(* This function block is responsible for holding the internal state of the function block that
   has the different tests in it (i.e. test-FB). Every test-FB can have one or more tests, and
   each test can do one or more asserts.
*)
{attribute 'call_after_init'}
{attribute 'reflection'}
FUNCTION_BLOCK FB_TestFunctionBlock IMPLEMENTS I_TestFunctionBlock
VAR
    {attribute 'instance-path'}
    {attribute 'noinit'}
    InstancePath : Tc2_Utilities.T_MaxString;

    (* This is a interface-pointer to the child-object that inherits this object
       in order for us to have a reference to calling the actual execution of the
       tests *) 
    RunnableTest : I_RunnableTestFunctionBlock;

    NumberOfTests : UINT := 0;
    TestNames : ARRAY[1..100] OF Tc2_Utilities.T_MaxString;
    TestFailed : ARRAY[1..100] OF BOOL;
END_VAR

METHOD PUBLIC AddTest
VAR_INPUT
    TestName : T_MaxString;
END_VAR
VAR
    CounterTestName : UINT;
END_VAR
(* Check if the test name already exists *)
FOR CounterTestName := 1 TO NumberOfTests BY 1 DO
    IF TestNames[CounterTestName] = TestName THEN
        RETURN; // Found
    END_IF
END_FOR

(* Not found. Add it. *)
TestNames[CounterTestName] := TestName;
NumberOfTests := NumberOfTests + 1;
END_METHOD

METHOD PUBLIC GetAmountOfFailedTests : UINT
VAR
    Counter : UINT;
    FailedTestsCount : UINT;
END_VAR
IF NumberOfTests > 0 THEN
    FOR Counter := 1 TO GetAmountOfTests() BY 1 DO
        IF TestFailed[Counter] = TRUE THEN
            FailedTestsCount := FailedTestsCount + 1;
        END_IF
    END_FOR
END_IF

GetAmountOfFailedTests := FailedTestsCount;
END_METHOD

METHOD PUBLIC GetAmountOfSuccessfulTests : UINT
GetAmountOfSuccessfulTests := GetAmountOfTests() - GetAmountOfFailedTests();
END_METHOD

METHOD PUBLIC GetAmountOfTests : UINT
GetAmountOfTests := NumberOfTests;
END_METHOD

METHOD PUBLIC GetInstancePath : Tc2_Utilities.T_MaxString
GetInstancePath := InstancePath;
END_METHOD

METHOD GetRunnable : I_RunnableTestFunctionBlock
GetRunnable := RunnableTest;
END_METHOD

{attribute 'call_after_init'}
METHOD PRIVATE Initialize
IF GVL.TestFunctionBlockAssertRegistered THEN
    GVL.AmountOfInitializedTestFunctionBlocks := GVL.AmountOfInitializedTestFunctionBlocks + 1;	
    GVL.TestFunctionBlockAddressess[GVL.AmountOfInitializedTestFunctionBlocks] := THIS^;
    GVL.TestFunctionBlockAssertRegistered := FALSE;
END_IF
END_METHOD

METHOD PUBLIC RegisterTestFunctionBlock
VAR_INPUT
	RunnableTestFunctionBlock : I_RunnableTestFunctionBlock;
END_VAR
RunnableTest := RunnableTestFunctionBlock;
END_METHOD

METHOD PUBLIC SetTestFailed
VAR_INPUT
    TestName : Tc2_Utilities.T_MaxString;
END_VAR
VAR
    Counter : UINT;
END_VAR
IF NumberOfTests > 0 THEN
    FOR Counter := 1 TO NumberOfTests BY 1 DO
        IF TestNames[Counter] = TestName THEN
            TestFailed[Counter] := TRUE;
        END_IF
    END_FOR
END_IF
END_METHOD

END_FUNCTION_BLOCK

(* stored: Version 1.1.0.1, ProductVersion 3.1.4022.12
   POU FB_TestFunctionBlock: Id {f80c23f2-119d-406b-ae11-06d1991bf64d}, SpecialFunc None
   Method AddTest: Id {d383011f-6bea-4b05-9018-ea4782ad2837}
   Method GetAmountOfFailedTests: Id {12e4522b-e67f-439a-af1d-8713231888aa}
   Method GetAmountOfSuccessfulTests: Id {635213dc-96ca-4be6-9c0d-c0454c29d34d}
   Method GetAmountOfTests: Id {6f67c6d5-c29e-4577-8651-51bd6db3ab63}
   Method GetInstancePath: Id {178fa338-5ed3-417b-8f4d-e9f120ace4b9}
   Method GetRunnable: Id {42018cb6-0640-401b-9af0-45a257049175}
   Method Initialize: Id {1c3645b8-e9b0-4963-8e9e-6ea2327dddf4}
   Method RegisterTestFunctionBlock: Id {5739bc4d-f91e-4513-b43f-1bc828337468}
   Method SetTestFailed: Id {79b1664f-2570-4cef-bd6e-d7307d9a7818} *)
